# EPICS substitutions: ATCACommonApp/Db/StreamUlong.substitutions
file "streamWf.db"  {
    pattern {      PORT,   DEVICE,  N,     TYPE,            DTYP,      FTVL,       NELM,    TSE      }
            { "$(PORT)", "$(DEV)",  0,  "ULONG", "asynInt32ArrayOut",   "ULONG",  "$(NELM)", "$(TSE)"    }
            { "$(PORT)", "$(DEV)",  1,  "ULONG", "asynInt32ArrayOut",   "ULONG",  "$(NELM)", "$(TSE)"    }
            { "$(PORT)", "$(DEV)",  2,  "ULONG", "asynInt32ArrayOut",   "ULONG",  "$(NELM)", "$(TSE)"    }
            { "$(PORT)", "$(DEV)",  3,  "ULONG", "asynInt32ArrayOut",   "ULONG",  "$(NELM)", "$(TSE)"    }

}
